FUNCTION_BLOCK EventWrapper_OLD (* Composite Function Block Type *)
  (* Standard: 61499-2 *)
  (* Version 0.0, 4/9/2019, erik, nxtControl GmbH, template *)
  PACKAGE Main;
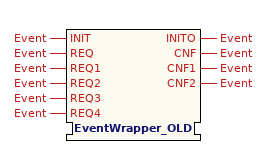
  EVENT_INPUT
    INIT; (* Initialization Request *)
    REQ; (* Normal Execution Request *)
    REQ1;
    REQ2;
    REQ3;
    REQ4;
  END_EVENT
  EVENT_OUTPUT
    INITO; (* Initialization Confirm *)
    CNF; (* Execution Confirmation *)
    CNF1;
    CNF2;
  END_EVENT
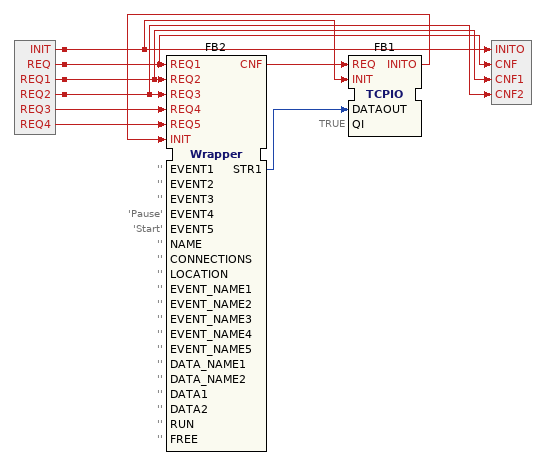
  FBS
    FB1 : TCPIO(QI := TRUE);
    FB2 : Wrapper(EVENT1 := '', EVENT2 := '', EVENT3 := '', EVENT4 := 'Pause', EVENT5 := 'Start', NAME := '', CONNECTIONS := '', LOCATION := '', EVENT_NAME1 := '', EVENT_NAME2 := '', EVENT_NAME3 := '', EVENT_NAME4 := '', EVENT_NAME5 := '', DATA_NAME1 := '', DATA_NAME2 := '', DATA1 := '', DATA2 := '', RUN := '', FREE := '');
  END_FBS
  EVENT_CONNECTIONS
    REQ TO FB2.REQ1;
    REQ1 TO FB2.REQ2;
    REQ2 TO FB2.REQ3;
    FB2.CNF TO FB1.REQ;
    REQ TO CNF;
    REQ1 TO CNF1;
    REQ2 TO CNF2;
    REQ3 TO FB2.REQ4;
    REQ4 TO FB2.REQ5;
    INIT TO FB1.INIT;
    FB1.INITO TO FB2.INIT;
    INIT TO INITO;
  END_CONNECTIONS
  DATA_CONNECTIONS
    FB2.STR1 TO FB1.DATAOUT;
  END_CONNECTIONS
END_FUNCTION_BLOCK
